TYPE ST_FcuControl :
STRUCT
	status	: ST_OpcuaStatus;
	
	input	: ST_FcuControl_in;	
	
	{attribute 'OPC.UA.DA.Access' := '1'}
	output	: ST_FcuControl_out;
END_STRUCT
END_TYPE

(* stored: Version 1.1.0.1, ProductVersion 3.1.4024.9
   DUT ST_FcuControl: Id {f4f7b709-9537-4936-8cb7-a1716639ff77} *)
